Universal Robots PolyScope program: Ejemplo_movimiento_relativo.urp

Program Ejemplo_movimiento_relativo (installation=default directory=/home/hugo/Documents/Proyecto_Ingenieria/ursim-5.10.2.106319/programs createdIn=5.10.2.106319 lastSavedIn=5.10.2.106319 robotSerialNumber=20195599999)
Calibrated DH parameters: a=[0, -0.425, -0.3922, 0, 0, 0]; d=[0.1625, 0, 0, 0.1333, 0.0997, 0.0996]; alpha=[1.570796, 0, 0, 1.570796, -1.570796, 0]; deltaTheta=[0, 0, 0, 0, 0, 0]
Robot Program (runOnlyOnce=false)
  MoveL speed 250 mm/s, acceleration 1200 mm/s^2 (useActiveTCP=true) feature=Base
    Waypoint Waypoint_1 (Relative): relativeFromPosition TCP in base x=490.93 y=300 z=200 mm, rx=-0.9946 ry=1.3694 rz=-1.0901 rad; joints [53.694, -136.544, -107.809, 63.332, 31.747, 14.323] deg; TCP in base x=490.93 y=500 z=200 mm, rx=-0.9946 ry=1.3694 rz=-1.0901 rad; joints [64.36, -147.67, -79.692, 45.868, 21.084, 14.848] deg
    Waypoint Waypoint_2 (Relative): relativeFromPosition TCP in base x=490.93 y=500 z=200 mm, rx=-0.9946 ry=1.3694 rz=-1.0901 rad; joints [64.36, -147.67, -79.692, 45.868, 21.084, 14.848] deg; TCP in base x=490.93 y=500 z=0 mm, rx=-0.9946 ry=1.3694 rz=-1.0901 rad; joints [64.36, -170.177, -68.136, 56.82, 21.084, 14.848] deg
    Waypoint Waypoint_3 (Relative): relativeFromPosition TCP in base x=490.93 y=500 z=0 mm, rx=-0.9946 ry=1.3694 rz=-1.0901 rad; joints [64.36, -170.177, -68.136, 56.82, 21.084, 14.848] deg; TCP in base x=490.93 y=300 z=0 mm, rx=-0.9946 ry=1.3694 rz=-1.0901 rad; joints [53.694, -162.992, -96.452, 78.423, 31.747, 14.323] deg
    Waypoint Waypoint_4 (Relative): relativeFromPosition TCP in base x=490.93 y=300 z=0 mm, rx=-0.9946 ry=1.3694 rz=-1.0901 rad; joints [53.694, -162.992, -96.452, 78.423, 31.747, 14.323] deg; TCP in base x=490.93 y=300 z=200 mm, rx=-0.9946 ry=1.3694 rz=-1.0901 rad; joints [53.694, -136.544, -107.809, 63.332, 31.747, 14.323] deg
